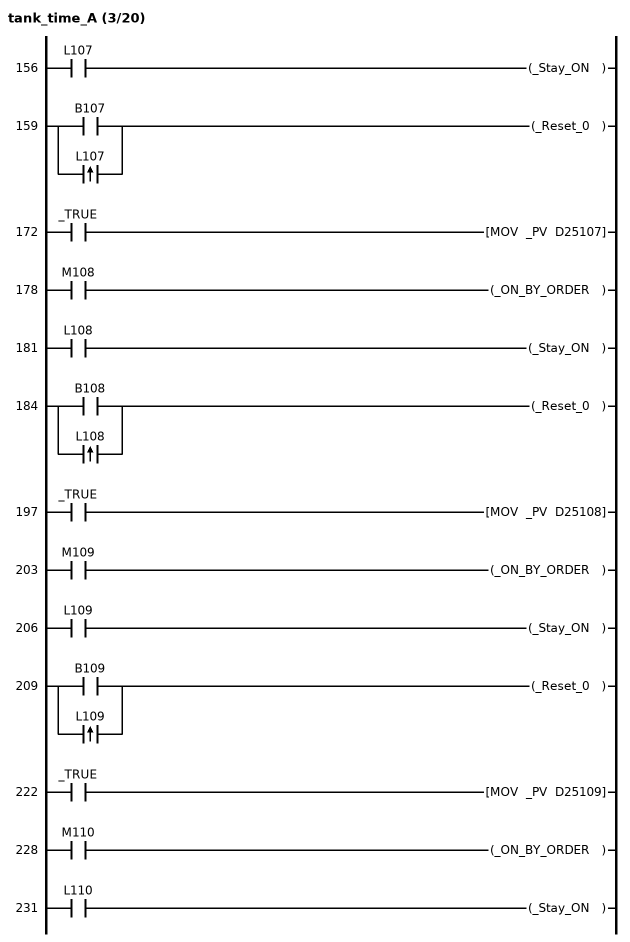
[picture p216: ladder of tank_time_A, rungs at steps 156 to 231]
156   LD      L107
      OUT     _Stay_ON
159   LD      B107
      ORP     L107
      OUT     _Reset_0
; FB START
; FB_NAME tank_PV
; INSTANCE_NAME tank_PV_7
; FB IN_B:ON_BY_ORDER
; FB OUT_PV:W
; FB IN_B:Stay_ON
; FB IN_B:Reset_0
; FB END
172   LD      _TRUE
      MOV     _PV D25107
; FB BLK END
; FB BLK START tank_PV(tank_PV_8)
178   LD      M108
      OUT     _ON_BY_ORDER
181   LD      L108
      OUT     _Stay_ON
184   LD      B108
      ORP     L108
      OUT     _Reset_0
; FB START
; FB_NAME tank_PV
; INSTANCE_NAME tank_PV_8
; FB IN_B:ON_BY_ORDER
; FB OUT_PV:W
; FB IN_B:Stay_ON
; FB IN_B:Reset_0
; FB END
197   LD      _TRUE
      MOV     _PV D25108
; FB BLK END
; FB BLK START tank_PV(tank_PV_9)
203   LD      M109
      OUT     _ON_BY_ORDER
206   LD      L109
      OUT     _Stay_ON
209   LD      B109
      ORP     L109
      OUT     _Reset_0
; FB START
; FB_NAME tank_PV
; INSTANCE_NAME tank_PV_9
; FB IN_B:ON_BY_ORDER
; FB OUT_PV:W
; FB IN_B:Stay_ON
; FB IN_B:Reset_0
; FB END
222   LD      _TRUE
      MOV     _PV D25109
; FB BLK END
; FB BLK START tank_PV(tank_PV_10)
228   LD      M110
      OUT     _ON_BY_ORDER
231   LD      L110
      OUT     _Stay_ON
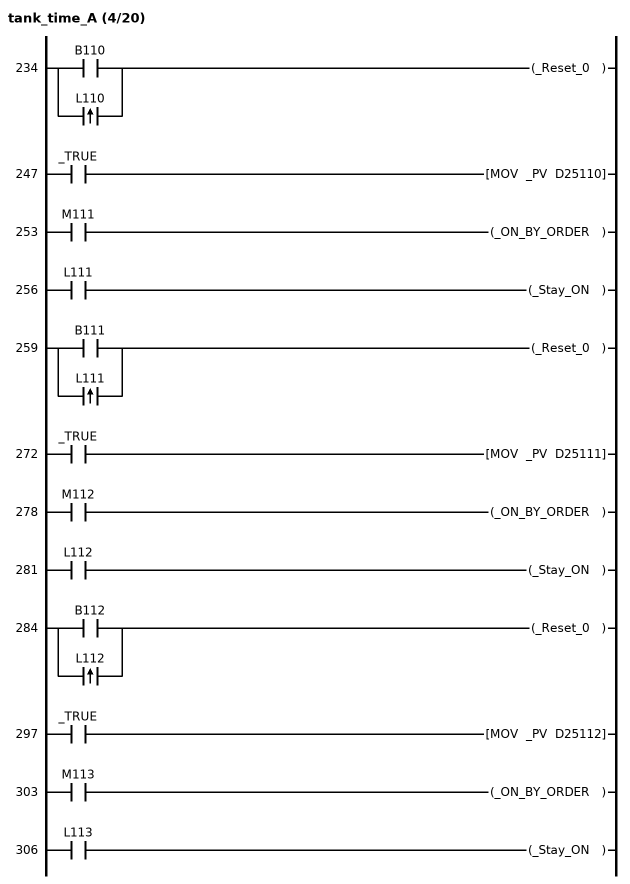
234   LD      B110
      ORP     L110
      OUT     _Reset_0
; FB START
; FB_NAME tank_PV
; INSTANCE_NAME tank_PV_10
; FB IN_B:ON_BY_ORDER
; FB OUT_PV:W
; FB IN_B:Stay_ON
; FB IN_B:Reset_0
; FB END
247   LD      _TRUE
      MOV     _PV D25110
; FB BLK END
; FB BLK START tank_PV(tank_PV_11)
253   LD      M111
      OUT     _ON_BY_ORDER
256   LD      L111
      OUT     _Stay_ON
259   LD      B111
      ORP     L111
      OUT     _Reset_0
; FB START
; FB_NAME tank_PV
; INSTANCE_NAME tank_PV_11
; FB IN_B:ON_BY_ORDER
; FB OUT_PV:W
; FB IN_B:Stay_ON
; FB IN_B:Reset_0
; FB END
272   LD      _TRUE
      MOV     _PV D25111
; FB BLK END
; FB BLK START tank_PV(tank_PV_12)
278   LD      M112
      OUT     _ON_BY_ORDER
281   LD      L112
      OUT     _Stay_ON
284   LD      B112
      ORP     L112
      OUT     _Reset_0
; FB START
; FB_NAME tank_PV
; INSTANCE_NAME tank_PV_12
; FB IN_B:ON_BY_ORDER
; FB OUT_PV:W
; FB IN_B:Stay_ON
; FB IN_B:Reset_0
; FB END
297   LD      _TRUE
      MOV     _PV D25112
; FB BLK END
; FB BLK START tank_PV(tank_PV_13)
303   LD      M113
      OUT     _ON_BY_ORDER
306   LD      L113
      OUT     _Stay_ON
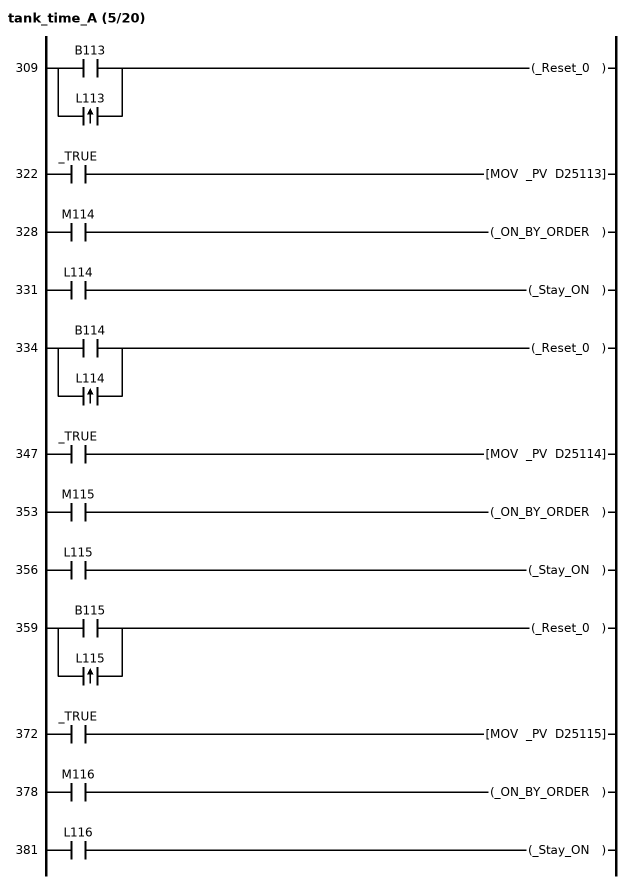
309   LD      B113
      ORP     L113
      OUT     _Reset_0
; FB START
; FB_NAME tank_PV
; INSTANCE_NAME tank_PV_13
; FB IN_B:ON_BY_ORDER
; FB OUT_PV:W
; FB IN_B:Stay_ON
; FB IN_B:Reset_0
; FB END
322   LD      _TRUE
      MOV     _PV D25113
; FB BLK END
; FB BLK START tank_PV(tank_PV_14)
328   LD      M114
      OUT     _ON_BY_ORDER
331   LD      L114
      OUT     _Stay_ON
334   LD      B114
      ORP     L114
      OUT     _Reset_0
; FB START
; FB_NAME tank_PV
; INSTANCE_NAME tank_PV_14
; FB IN_B:ON_BY_ORDER
; FB OUT_PV:W
; FB IN_B:Stay_ON
; FB IN_B:Reset_0
; FB END
347   LD      _TRUE
      MOV     _PV D25114
; FB BLK END
; FB BLK START tank_PV(tank_PV_15)
353   LD      M115
      OUT     _ON_BY_ORDER
356   LD      L115
      OUT     _Stay_ON
359   LD      B115
      ORP     L115
      OUT     _Reset_0
; FB START
; FB_NAME tank_PV
; INSTANCE_NAME tank_PV_15
; FB IN_B:ON_BY_ORDER
; FB OUT_PV:W
; FB IN_B:Stay_ON
; FB IN_B:Reset_0
; FB END
372   LD      _TRUE
      MOV     _PV D25115
; FB BLK END
; FB BLK START tank_PV(tank_PV_16)
378   LD      M116
      OUT     _ON_BY_ORDER
381   LD      L116
      OUT     _Stay_ON
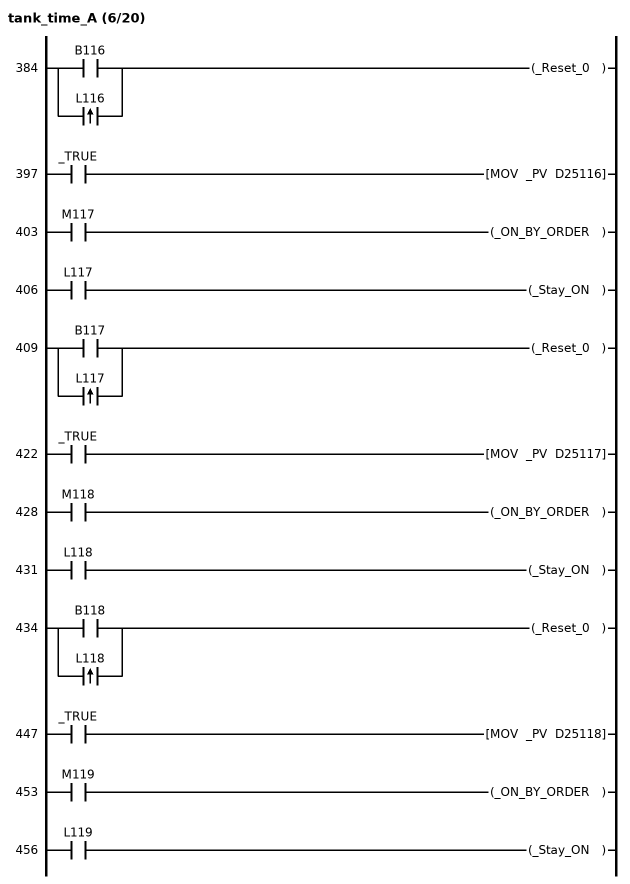
384   LD      B116
      ORP     L116
      OUT     _Reset_0
; FB START
; FB_NAME tank_PV
; INSTANCE_NAME tank_PV_16
; FB IN_B:ON_BY_ORDER
; FB OUT_PV:W
; FB IN_B:Stay_ON
; FB IN_B:Reset_0
; FB END
397   LD      _TRUE
      MOV     _PV D25116
; FB BLK END
; FB BLK START tank_PV(tank_PV_17)
403   LD      M117
      OUT     _ON_BY_ORDER
406   LD      L117
      OUT     _Stay_ON
409   LD      B117
      ORP     L117
      OUT     _Reset_0
; FB START
; FB_NAME tank_PV
; INSTANCE_NAME tank_PV_17
; FB IN_B:ON_BY_ORDER
; FB OUT_PV:W
; FB IN_B:Stay_ON
; FB IN_B:Reset_0
; FB END
422   LD      _TRUE
      MOV     _PV D25117
; FB BLK END
; FB BLK START tank_PV(tank_PV_18)
428   LD      M118
      OUT     _ON_BY_ORDER
431   LD      L118
      OUT     _Stay_ON
434   LD      B118
      ORP     L118
      OUT     _Reset_0
; FB START
; FB_NAME tank_PV
; INSTANCE_NAME tank_PV_18
; FB IN_B:ON_BY_ORDER
; FB OUT_PV:W
; FB IN_B:Stay_ON
; FB IN_B:Reset_0
; FB END
447   LD      _TRUE
      MOV     _PV D25118
; FB BLK END
; FB BLK START tank_PV(tank_PV_19)
453   LD      M119
      OUT     _ON_BY_ORDER
456   LD      L119
      OUT     _Stay_ON
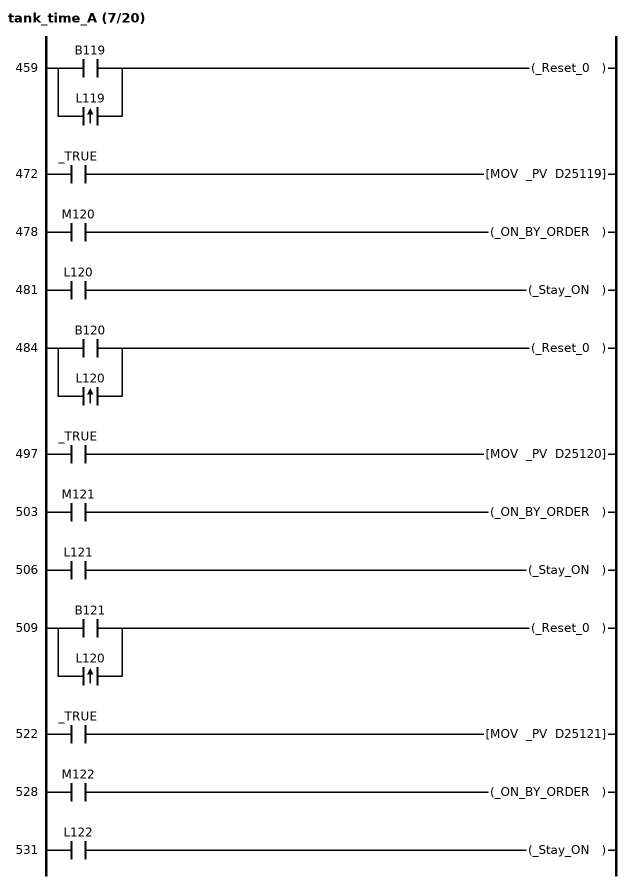
459   LD      B119
      ORP     L119
      OUT     _Reset_0
; FB START
; FB_NAME tank_PV
; INSTANCE_NAME tank_PV_19
; FB IN_B:ON_BY_ORDER
; FB OUT_PV:W
; FB IN_B:Stay_ON
; FB IN_B:Reset_0
; FB END
472   LD      _TRUE
      MOV     _PV D25119
; FB BLK END
; FB BLK START tank_PV(tank_PV_20)
478   LD      M120
      OUT     _ON_BY_ORDER
481   LD      L120
      OUT     _Stay_ON
484   LD      B120
      ORP     L120
      OUT     _Reset_0
; FB START
; FB_NAME tank_PV
; INSTANCE_NAME tank_PV_20
; FB IN_B:ON_BY_ORDER
; FB OUT_PV:W
; FB IN_B:Stay_ON
; FB IN_B:Reset_0
; FB END
497   LD      _TRUE
      MOV     _PV D25120
; FB BLK END
; FB BLK START tank_PV(tank_PV_21)
503   LD      M121
      OUT     _ON_BY_ORDER
506   LD      L121
      OUT     _Stay_ON
509   LD      B121
      ORP     L120
      OUT     _Reset_0
; FB START
; FB_NAME tank_PV
; INSTANCE_NAME tank_PV_21
; FB IN_B:ON_BY_ORDER
; FB OUT_PV:W
; FB IN_B:Stay_ON
; FB IN_B:Reset_0
; FB END
522   LD      _TRUE
      MOV     _PV D25121
; FB BLK END
; FB BLK START tank_PV(tank_PV_22)
528   LD      M122
      OUT     _ON_BY_ORDER
531   LD      L122
      OUT     _Stay_ON
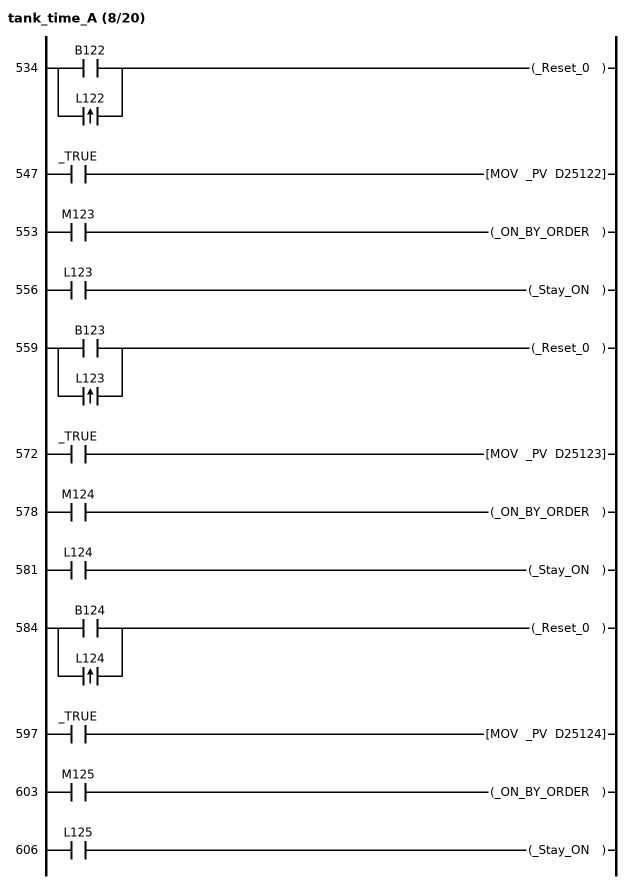
534   LD      B122
      ORP     L122
      OUT     _Reset_0
; FB START
; FB_NAME tank_PV
; INSTANCE_NAME tank_PV_22
; FB IN_B:ON_BY_ORDER
; FB OUT_PV:W
; FB IN_B:Stay_ON
; FB IN_B:Reset_0
; FB END
547   LD      _TRUE
      MOV     _PV D25122
; FB BLK END
; FB BLK START tank_PV(tank_PV_23)
553   LD      M123
      OUT     _ON_BY_ORDER
556   LD      L123
      OUT     _Stay_ON
559   LD      B123
      ORP     L123
      OUT     _Reset_0
; FB START
; FB_NAME tank_PV
; INSTANCE_NAME tank_PV_23
; FB IN_B:ON_BY_ORDER
; FB OUT_PV:W
; FB IN_B:Stay_ON
; FB IN_B:Reset_0
; FB END
572   LD      _TRUE
      MOV     _PV D25123
; FB BLK END
; FB BLK START tank_PV(tank_PV_24)
578   LD      M124
      OUT     _ON_BY_ORDER
581   LD      L124
      OUT     _Stay_ON
584   LD      B124
      ORP     L124
      OUT     _Reset_0
; FB START
; FB_NAME tank_PV
; INSTANCE_NAME tank_PV_24
; FB IN_B:ON_BY_ORDER
; FB OUT_PV:W
; FB IN_B:Stay_ON
; FB IN_B:Reset_0
; FB END
597   LD      _TRUE
      MOV     _PV D25124
; FB BLK END
; FB BLK START tank_PV(tank_PV_25)
603   LD      M125
      OUT     _ON_BY_ORDER
606   LD      L125
      OUT     _Stay_ON
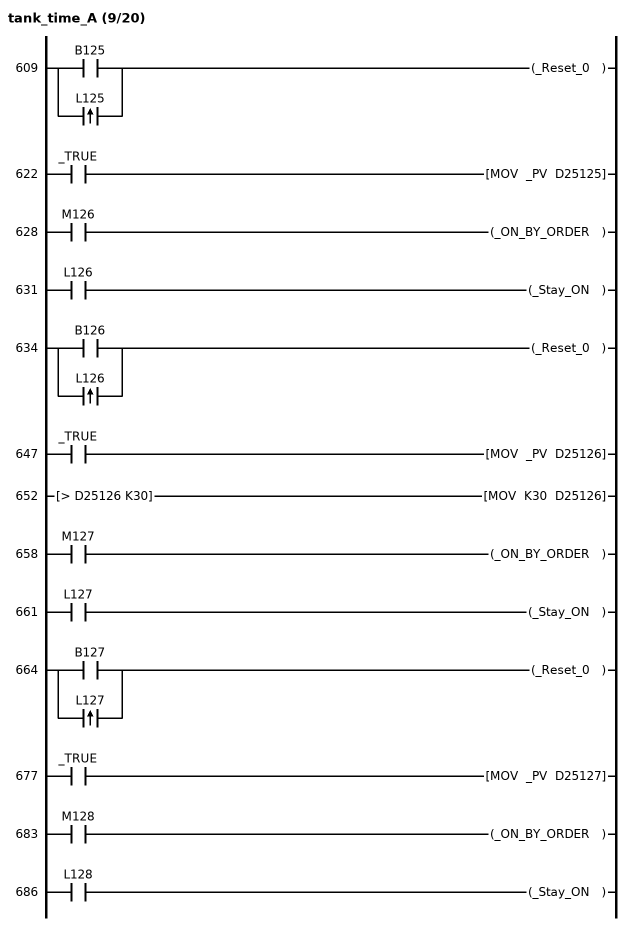
609   LD      B125
      ORP     L125
      OUT     _Reset_0
; FB START
; FB_NAME tank_PV
; INSTANCE_NAME tank_PV_25
; FB IN_B:ON_BY_ORDER
; FB OUT_PV:W
; FB IN_B:Stay_ON
; FB IN_B:Reset_0
; FB END
622   LD      _TRUE
      MOV     _PV D25125
; FB BLK END
; FB BLK START tank_PV(tank_PV_26)
628   LD      M126
      OUT     _ON_BY_ORDER
631   LD      L126
      OUT     _Stay_ON
634   LD      B126
      ORP     L126
      OUT     _Reset_0
; FB START
; FB_NAME tank_PV
; INSTANCE_NAME tank_PV_26
; FB IN_B:ON_BY_ORDER
; FB OUT_PV:W
; FB IN_B:Stay_ON
; FB IN_B:Reset_0
; FB END
647   LD      _TRUE
      MOV     _PV D25126
; FB BLK END
652   LD>     D25126 K30
      MOV     K30 D25126
; FB BLK START tank_PV(tank_PV_27)
658   LD      M127
      OUT     _ON_BY_ORDER
661   LD      L127
      OUT     _Stay_ON
664   LD      B127
      ORP     L127
      OUT     _Reset_0
; FB START
; FB_NAME tank_PV
; INSTANCE_NAME tank_PV_27
; FB IN_B:ON_BY_ORDER
; FB OUT_PV:W
; FB IN_B:Stay_ON
; FB IN_B:Reset_0
; FB END
677   LD      _TRUE
      MOV     _PV D25127
; FB BLK END
; FB BLK START tank_PV(tank_PV_28)
683   LD      M128
      OUT     _ON_BY_ORDER
686   LD      L128
      OUT     _Stay_ON
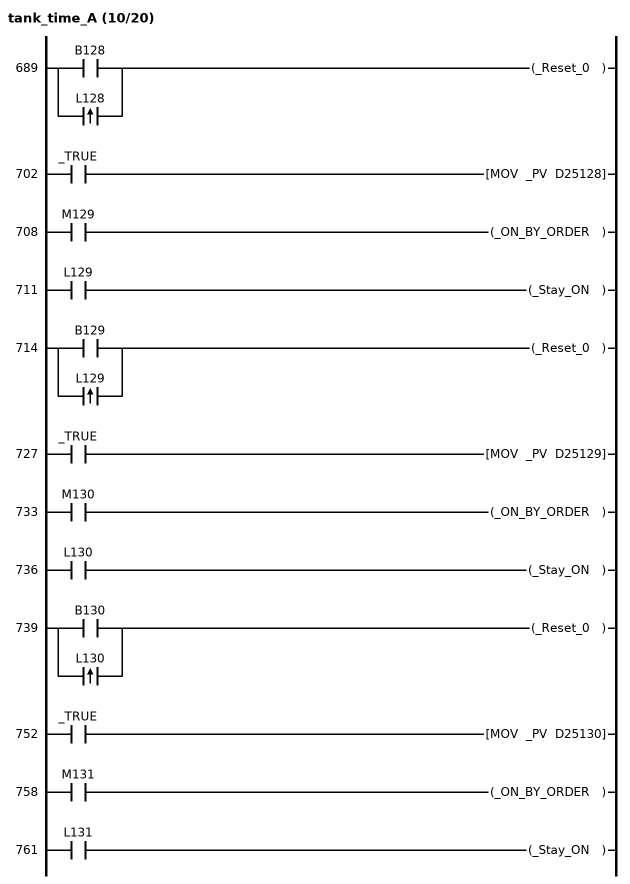
689   LD      B128
      ORP     L128
      OUT     _Reset_0
; FB START
; FB_NAME tank_PV
; INSTANCE_NAME tank_PV_28
; FB IN_B:ON_BY_ORDER
; FB OUT_PV:W
; FB IN_B:Stay_ON
; FB IN_B:Reset_0
; FB END
702   LD      _TRUE
      MOV     _PV D25128
; FB BLK END
; FB BLK START tank_PV(tank_PV_29)
708   LD      M129
      OUT     _ON_BY_ORDER
711   LD      L129
      OUT     _Stay_ON
714   LD      B129
      ORP     L129
      OUT     _Reset_0
; FB START
; FB_NAME tank_PV
; INSTANCE_NAME tank_PV_29
; FB IN_B:ON_BY_ORDER
; FB OUT_PV:W
; FB IN_B:Stay_ON
; FB IN_B:Reset_0
; FB END
727   LD      _TRUE
      MOV     _PV D25129
; FB BLK END
; FB BLK START tank_PV(tank_PV_30)
733   LD      M130
      OUT     _ON_BY_ORDER
736   LD      L130
      OUT     _Stay_ON
739   LD      B130
      ORP     L130
      OUT     _Reset_0
; FB START
; FB_NAME tank_PV
; INSTANCE_NAME tank_PV_30
; FB IN_B:ON_BY_ORDER
; FB OUT_PV:W
; FB IN_B:Stay_ON
; FB IN_B:Reset_0
; FB END
752   LD      _TRUE
      MOV     _PV D25130
; FB BLK END
; FB BLK START tank_PV(tank_PV_31)
758   LD      M131
      OUT     _ON_BY_ORDER
761   LD      L131
      OUT     _Stay_ON
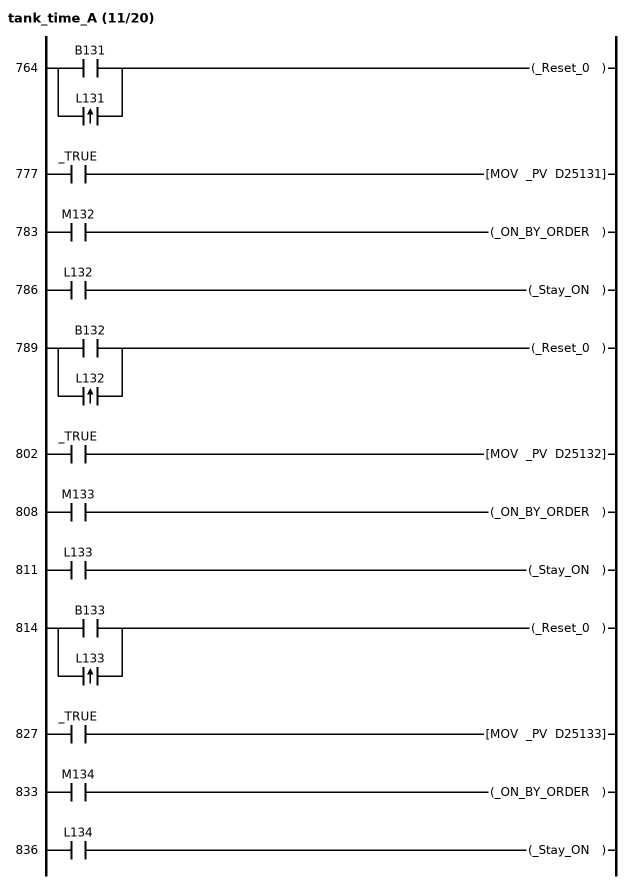
764   LD      B131
      ORP     L131
      OUT     _Reset_0
; FB START
; FB_NAME tank_PV
; INSTANCE_NAME tank_PV_31
; FB IN_B:ON_BY_ORDER
; FB OUT_PV:W
; FB IN_B:Stay_ON
; FB IN_B:Reset_0
; FB END
777   LD      _TRUE
      MOV     _PV D25131
; FB BLK END
; FB BLK START tank_PV(tank_PV_32)
783   LD      M132
      OUT     _ON_BY_ORDER
786   LD      L132
      OUT     _Stay_ON
789   LD      B132
      ORP     L132
      OUT     _Reset_0
; FB START
; FB_NAME tank_PV
; INSTANCE_NAME tank_PV_32
; FB IN_B:ON_BY_ORDER
; FB OUT_PV:W
; FB IN_B:Stay_ON
; FB IN_B:Reset_0
; FB END
802   LD      _TRUE
      MOV     _PV D25132
; FB BLK END
; FB BLK START tank_PV(tank_PV_33)
808   LD      M133
      OUT     _ON_BY_ORDER
811   LD      L133
      OUT     _Stay_ON
814   LD      B133
      ORP     L133
      OUT     _Reset_0
; FB START
; FB_NAME tank_PV
; INSTANCE_NAME tank_PV_33
; FB IN_B:ON_BY_ORDER
; FB OUT_PV:W
; FB IN_B:Stay_ON
; FB IN_B:Reset_0
; FB END
827   LD      _TRUE
      MOV     _PV D25133
; FB BLK END
; FB BLK START tank_PV(tank_PV_34)
833   LD      M134
      OUT     _ON_BY_ORDER
836   LD      L134
      OUT     _Stay_ON
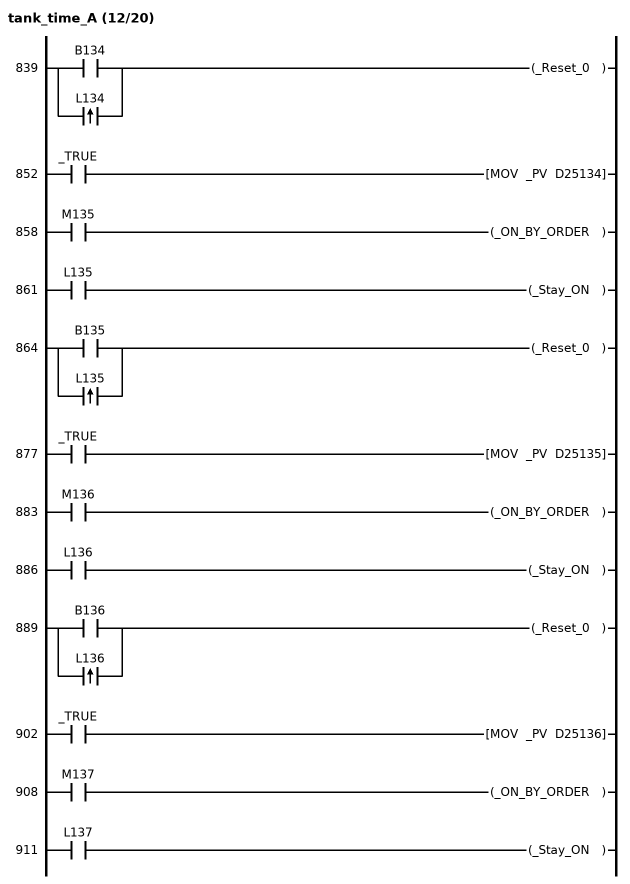
839   LD      B134
      ORP     L134
      OUT     _Reset_0
; FB START
; FB_NAME tank_PV
; INSTANCE_NAME tank_PV_34
; FB IN_B:ON_BY_ORDER
; FB OUT_PV:W
; FB IN_B:Stay_ON
; FB IN_B:Reset_0
; FB END
852   LD      _TRUE
      MOV     _PV D25134
; FB BLK END
; FB BLK START tank_PV(tank_PV_35)
858   LD      M135
      OUT     _ON_BY_ORDER
861   LD      L135
      OUT     _Stay_ON
864   LD      B135
      ORP     L135
      OUT     _Reset_0
; FB START
; FB_NAME tank_PV
; INSTANCE_NAME tank_PV_35
; FB IN_B:ON_BY_ORDER
; FB OUT_PV:W
; FB IN_B:Stay_ON
; FB IN_B:Reset_0
; FB END
877   LD      _TRUE
      MOV     _PV D25135
; FB BLK END
; FB BLK START tank_PV(tank_PV_36)
883   LD      M136
      OUT     _ON_BY_ORDER
886   LD      L136
      OUT     _Stay_ON
889   LD      B136
      ORP     L136
      OUT     _Reset_0
; FB START
; FB_NAME tank_PV
; INSTANCE_NAME tank_PV_36
; FB IN_B:ON_BY_ORDER
; FB OUT_PV:W
; FB IN_B:Stay_ON
; FB IN_B:Reset_0
; FB END
902   LD      _TRUE
      MOV     _PV D25136
; FB BLK END
; FB BLK START tank_PV(tank_PV_37)
908   LD      M137
      OUT     _ON_BY_ORDER
911   LD      L137
      OUT     _Stay_ON
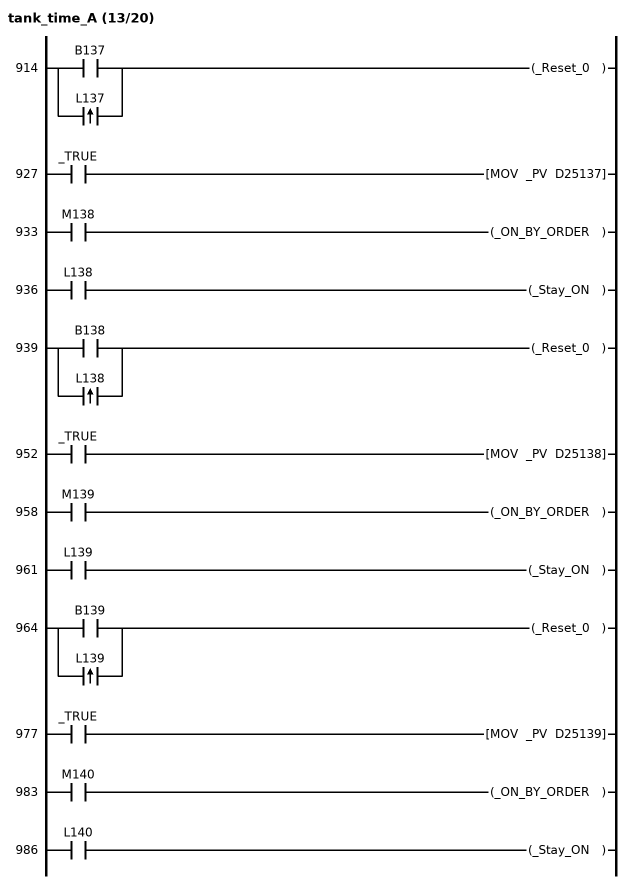
914   LD      B137
      ORP     L137
      OUT     _Reset_0
; FB START
; FB_NAME tank_PV
; INSTANCE_NAME tank_PV_37
; FB IN_B:ON_BY_ORDER
; FB OUT_PV:W
; FB IN_B:Stay_ON
; FB IN_B:Reset_0
; FB END
927   LD      _TRUE
      MOV     _PV D25137
; FB BLK END
; FB BLK START tank_PV(tank_PV_38)
933   LD      M138
      OUT     _ON_BY_ORDER
936   LD      L138
      OUT     _Stay_ON
939   LD      B138
      ORP     L138
      OUT     _Reset_0
; FB START
; FB_NAME tank_PV
; INSTANCE_NAME tank_PV_38
; FB IN_B:ON_BY_ORDER
; FB OUT_PV:W
; FB IN_B:Stay_ON
; FB IN_B:Reset_0
; FB END
952   LD      _TRUE
      MOV     _PV D25138
; FB BLK END
; FB BLK START tank_PV(tank_PV_39)
958   LD      M139
      OUT     _ON_BY_ORDER
961   LD      L139
      OUT     _Stay_ON
964   LD      B139
      ORP     L139
      OUT     _Reset_0
; FB START
; FB_NAME tank_PV
; INSTANCE_NAME tank_PV_39
; FB IN_B:ON_BY_ORDER
; FB OUT_PV:W
; FB IN_B:Stay_ON
; FB IN_B:Reset_0
; FB END
977   LD      _TRUE
      MOV     _PV D25139
; FB BLK END
; FB BLK START tank_PV(tank_PV_40)
983   LD      M140
      OUT     _ON_BY_ORDER
986   LD      L140
      OUT     _Stay_ON
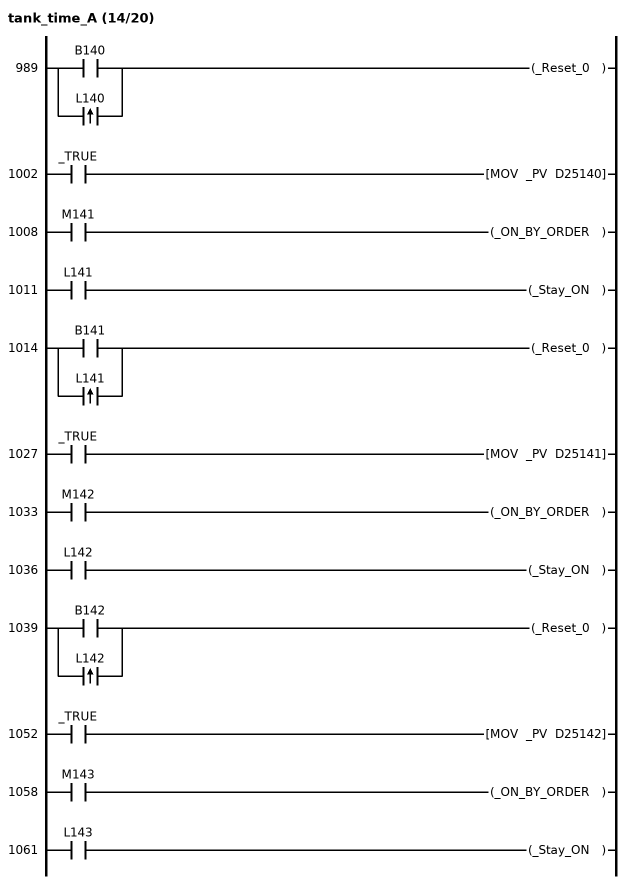
989   LD      B140
      ORP     L140
      OUT     _Reset_0
; FB START
; FB_NAME tank_PV
; INSTANCE_NAME tank_PV_40
; FB IN_B:ON_BY_ORDER
; FB OUT_PV:W
; FB IN_B:Stay_ON
; FB IN_B:Reset_0
; FB END
1002  LD      _TRUE
      MOV     _PV D25140
; FB BLK END
; FB BLK START tank_PV(tank_PV_41)
1008  LD      M141
      OUT     _ON_BY_ORDER
1011  LD      L141
      OUT     _Stay_ON
1014  LD      B141
      ORP     L141
      OUT     _Reset_0
; FB START
; FB_NAME tank_PV
; INSTANCE_NAME tank_PV_41
; FB IN_B:ON_BY_ORDER
; FB OUT_PV:W
; FB IN_B:Stay_ON
; FB IN_B:Reset_0
; FB END
1027  LD      _TRUE
      MOV     _PV D25141
; FB BLK END
; FB BLK START tank_PV(tank_PV_42)
1033  LD      M142
      OUT     _ON_BY_ORDER
1036  LD      L142
      OUT     _Stay_ON
1039  LD      B142
      ORP     L142
      OUT     _Reset_0
; FB START
; FB_NAME tank_PV
; INSTANCE_NAME tank_PV_42
; FB IN_B:ON_BY_ORDER
; FB OUT_PV:W
; FB IN_B:Stay_ON
; FB IN_B:Reset_0
; FB END
1052  LD      _TRUE
      MOV     _PV D25142
; FB BLK END
; FB BLK START tank_PV(tank_PV_43)
1058  LD      M143
      OUT     _ON_BY_ORDER
1061  LD      L143
      OUT     _Stay_ON
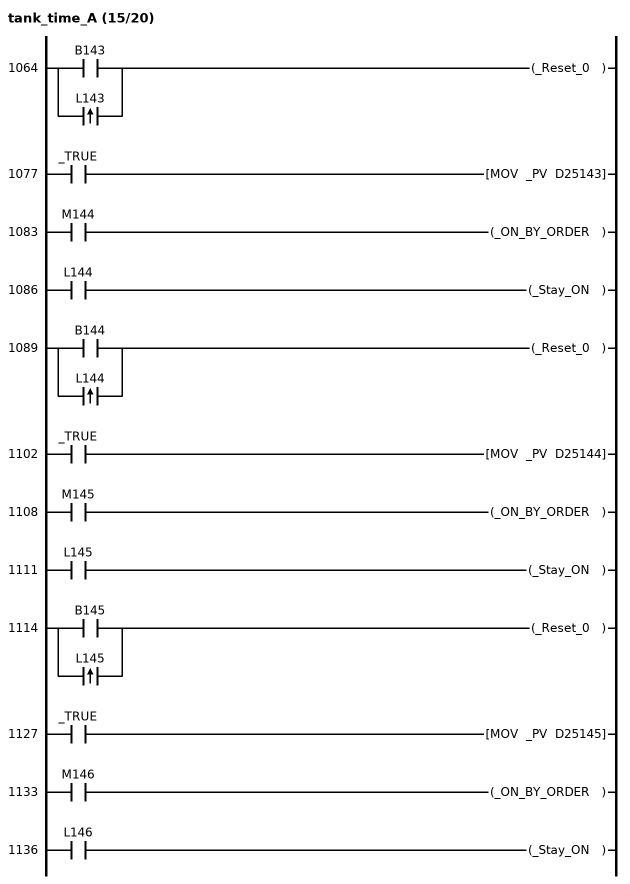
1064  LD      B143
      ORP     L143
      OUT     _Reset_0
; FB START
; FB_NAME tank_PV
; INSTANCE_NAME tank_PV_43
; FB IN_B:ON_BY_ORDER
; FB OUT_PV:W
; FB IN_B:Stay_ON
; FB IN_B:Reset_0
; FB END
1077  LD      _TRUE
      MOV     _PV D25143
; FB BLK END
; FB BLK START tank_PV(tank_PV_44)
1083  LD      M144
      OUT     _ON_BY_ORDER
1086  LD      L144
      OUT     _Stay_ON
1089  LD      B144
      ORP     L144
      OUT     _Reset_0
; FB START
; FB_NAME tank_PV
; INSTANCE_NAME tank_PV_44
; FB IN_B:ON_BY_ORDER
; FB OUT_PV:W
; FB IN_B:Stay_ON
; FB IN_B:Reset_0
; FB END
1102  LD      _TRUE
      MOV     _PV D25144
; FB BLK END
; FB BLK START tank_PV(tank_PV_45)
1108  LD      M145
      OUT     _ON_BY_ORDER
1111  LD      L145
      OUT     _Stay_ON
1114  LD      B145
      ORP     L145
      OUT     _Reset_0
; FB START
; FB_NAME tank_PV
; INSTANCE_NAME tank_PV_45
; FB IN_B:ON_BY_ORDER
; FB OUT_PV:W
; FB IN_B:Stay_ON
; FB IN_B:Reset_0
; FB END
1127  LD      _TRUE
      MOV     _PV D25145
; FB BLK END
; FB BLK START tank_PV(tank_PV_46)
1133  LD      M146
      OUT     _ON_BY_ORDER
1136  LD      L146
      OUT     _Stay_ON
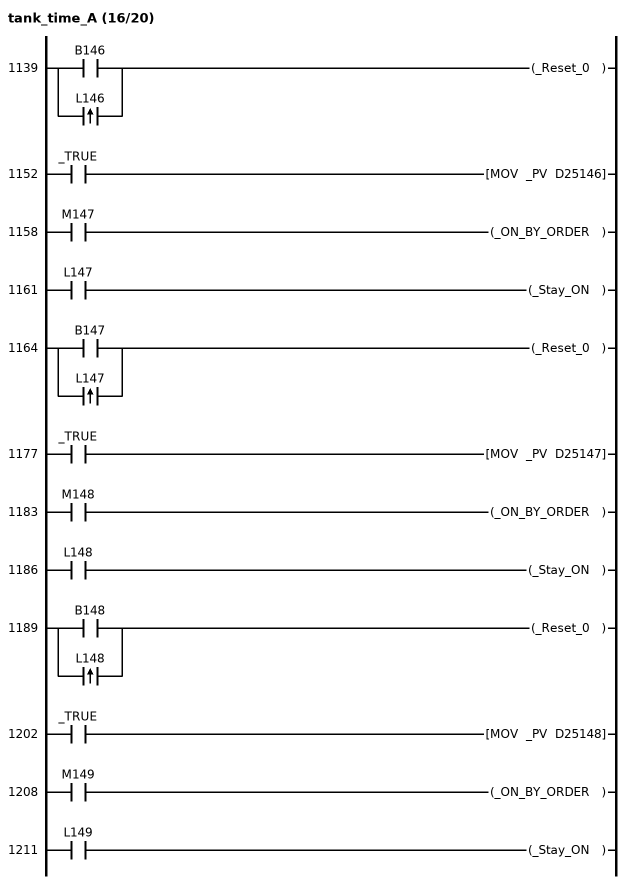
1139  LD      B146
      ORP     L146
      OUT     _Reset_0
; FB START
; FB_NAME tank_PV
; INSTANCE_NAME tank_PV_46
; FB IN_B:ON_BY_ORDER
; FB OUT_PV:W
; FB IN_B:Stay_ON
; FB IN_B:Reset_0
; FB END
1152  LD      _TRUE
      MOV     _PV D25146
; FB BLK END
; FB BLK START tank_PV(tank_PV_47)
1158  LD      M147
      OUT     _ON_BY_ORDER
1161  LD      L147
      OUT     _Stay_ON
1164  LD      B147
      ORP     L147
      OUT     _Reset_0
; FB START
; FB_NAME tank_PV
; INSTANCE_NAME tank_PV_47
; FB IN_B:ON_BY_ORDER
; FB OUT_PV:W
; FB IN_B:Stay_ON
; FB IN_B:Reset_0
; FB END
1177  LD      _TRUE
      MOV     _PV D25147
; FB BLK END
; FB BLK START tank_PV(tank_PV_48)
1183  LD      M148
      OUT     _ON_BY_ORDER
1186  LD      L148
      OUT     _Stay_ON
1189  LD      B148
      ORP     L148
      OUT     _Reset_0
; FB START
; FB_NAME tank_PV
; INSTANCE_NAME tank_PV_48
; FB IN_B:ON_BY_ORDER
; FB OUT_PV:W
; FB IN_B:Stay_ON
; FB IN_B:Reset_0
; FB END
1202  LD      _TRUE
      MOV     _PV D25148
; FB BLK END
; FB BLK START tank_PV(tank_PV_49)
1208  LD      M149
      OUT     _ON_BY_ORDER
1211  LD      L149
      OUT     _Stay_ON
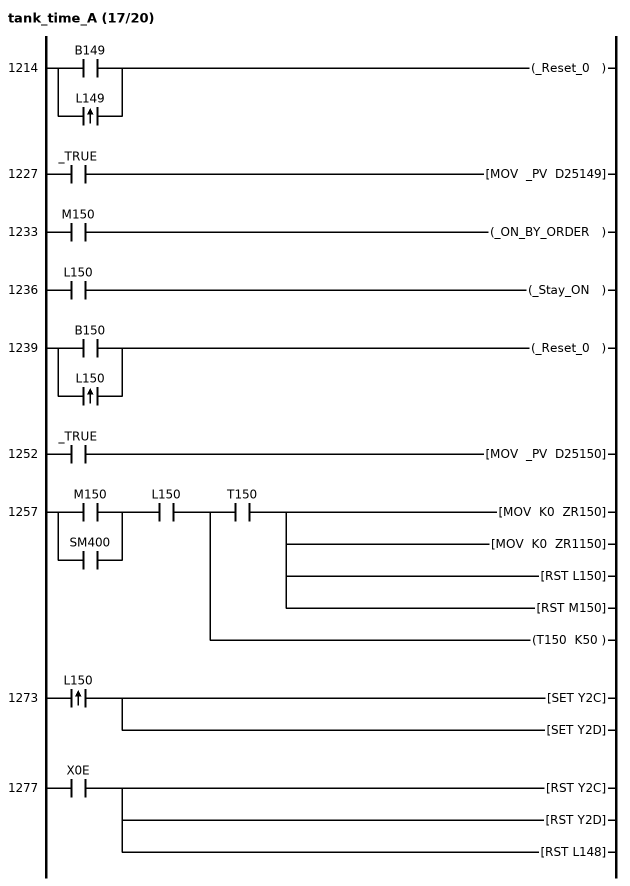
1214  LD      B149
      ORP     L149
      OUT     _Reset_0
; FB START
; FB_NAME tank_PV
; INSTANCE_NAME tank_PV_49
; FB IN_B:ON_BY_ORDER
; FB OUT_PV:W
; FB IN_B:Stay_ON
; FB IN_B:Reset_0
; FB END
1227  LD      _TRUE
      MOV     _PV D25149
; FB BLK END
; FB BLK START tank_PV(tank_PV_50)
1233  LD      M150
      OUT     _ON_BY_ORDER
1236  LD      L150
      OUT     _Stay_ON
1239  LD      B150
      ORP     L150
      OUT     _Reset_0
; FB START
; FB_NAME tank_PV
; INSTANCE_NAME tank_PV_50
; FB IN_B:ON_BY_ORDER
; FB OUT_PV:W
; FB IN_B:Stay_ON
; FB IN_B:Reset_0
; FB END
1252  LD      _TRUE
      MOV     _PV D25150
; FB BLK END
1257  LD      M150
      OR      SM400
      AND     L150
      MPS
      AND     T150
      MOV     K0 ZR150
      MOV     K0 ZR1150
      RST     L150
      RST     M150
      MPP
      OUT     T150 K50
1273  LDP     L150
      SET     Y2C
      SET     Y2D
1277  LD      X0E
      RST     Y2C
      RST     Y2D
      RST     L148
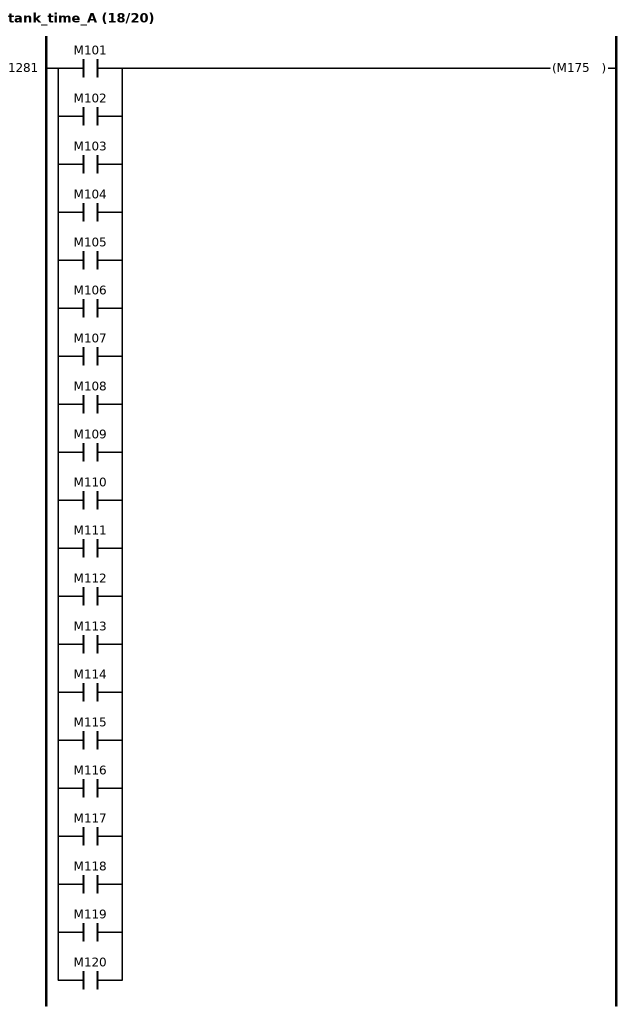
1281  LD      M101
      OR      M102
      OR      M103
      OR      M104
      OR      M105
      OR      M106
      OR      M107
      OR      M108
      OR      M109
      OR      M110
      OR      M111
      OR      M112
      OR      M113
      OR      M114
      OR      M115
      OR      M116
      OR      M117
      OR      M118
      OR      M119
      OR      M120
      OUT     M175
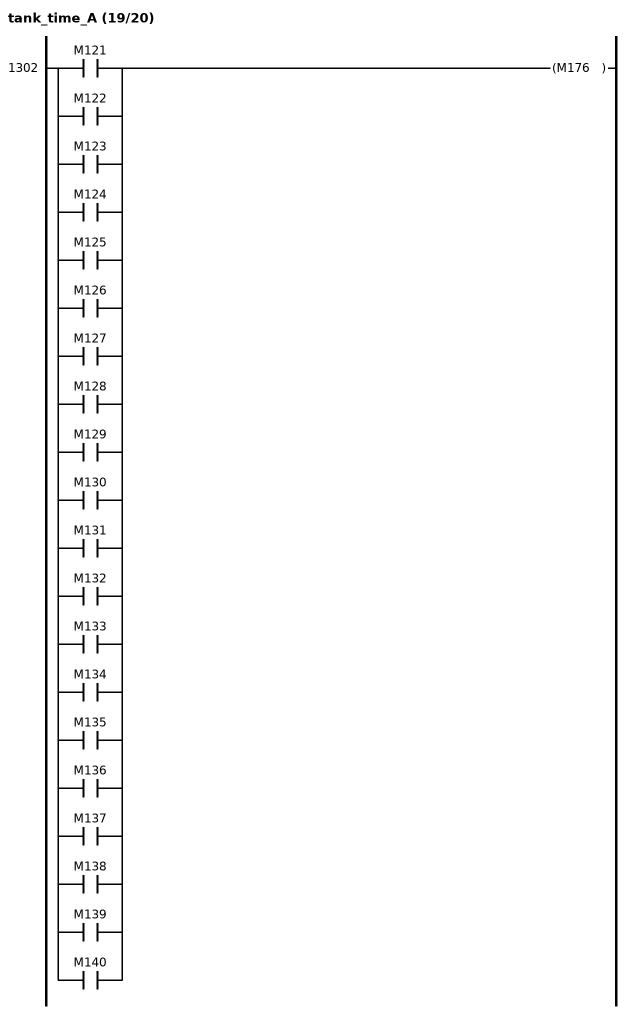
1302  LD      M121
      OR      M122
      OR      M123
      OR      M124
      OR      M125
      OR      M126
      OR      M127
      OR      M128
      OR      M129
      OR      M130
      OR      M131
      OR      M132
      OR      M133
      OR      M134
      OR      M135
      OR      M136
      OR      M137
      OR      M138
      OR      M139
      OR      M140
      OUT     M176
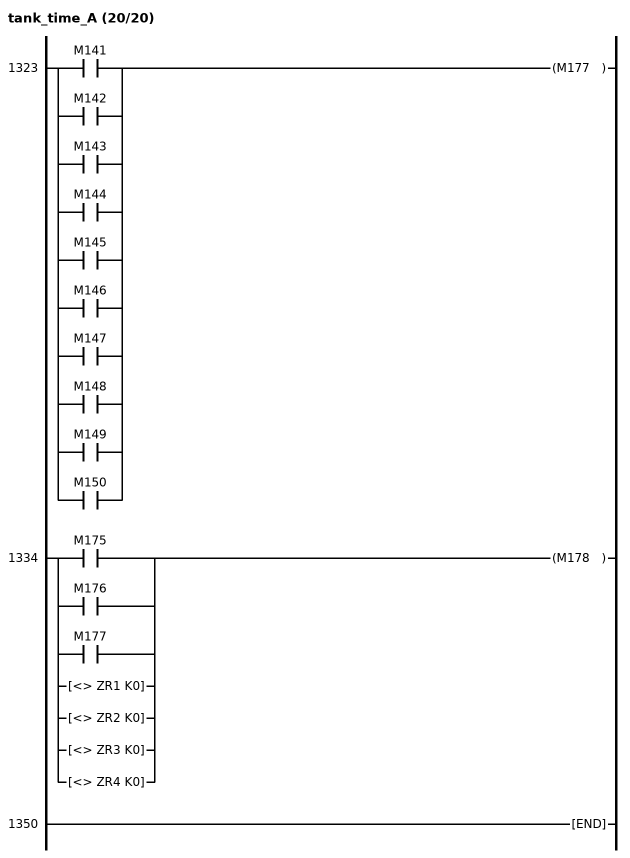
1323  LD      M141
      OR      M142
      OR      M143
      OR      M144
      OR      M145
      OR      M146
      OR      M147
      OR      M148
      OR      M149
      OR      M150
      OUT     M177
1334  LD      M175
      OR      M176
      OR      M177
      OR<>    ZR1 K0
      OR<>    ZR2 K0
      OR<>    ZR3 K0
      OR<>    ZR4 K0
      OUT     M178
1350  END
END_PROGRAM

PROGRAM temp_system
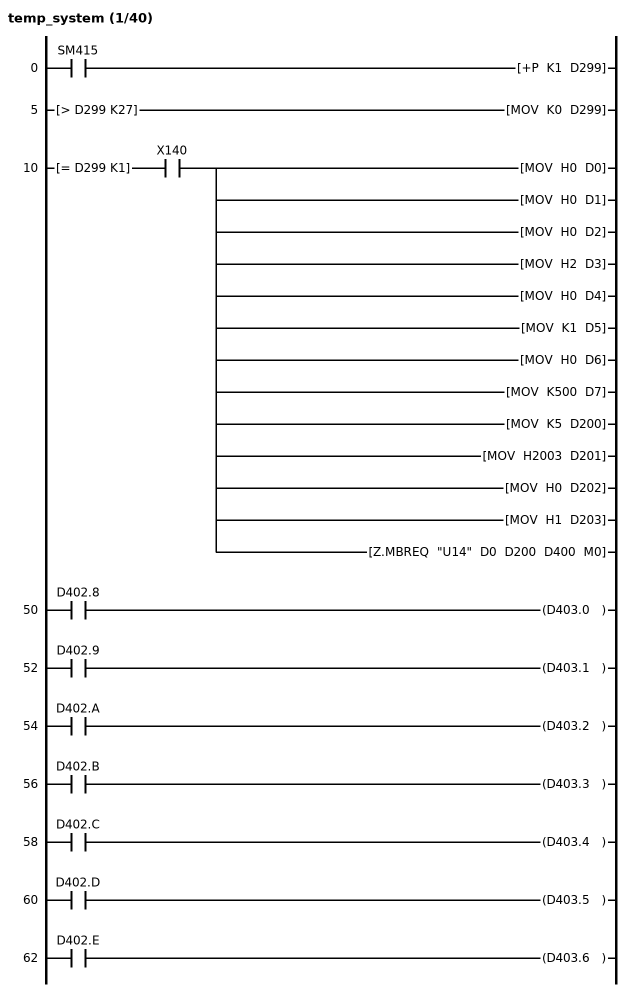
0     LD      SM415
      +P      K1 D299
5     LD>     D299 K27
      MOV     K0 D299
10    LD=     D299 K1
      AND     X140
      MOV     H0 D0
      MOV     H0 D1
      MOV     H0 D2
      MOV     H2 D3
      MOV     H0 D4
      MOV     K1 D5
      MOV     H0 D6
      MOV     K500 D7
      MOV     K5 D200
      MOV     H2003 D201
      MOV     H0 D202
      MOV     H1 D203
      Z.MBREQ "U14" D0 D200 D400 M0
50    LD      D402.8
      OUT     D403.0
52    LD      D402.9
      OUT     D403.1
54    LD      D402.A
      OUT     D403.2
56    LD      D402.B
      OUT     D403.3
58    LD      D402.C
      OUT     D403.4
60    LD      D402.D
      OUT     D403.5
62    LD      D402.E
      OUT     D403.6
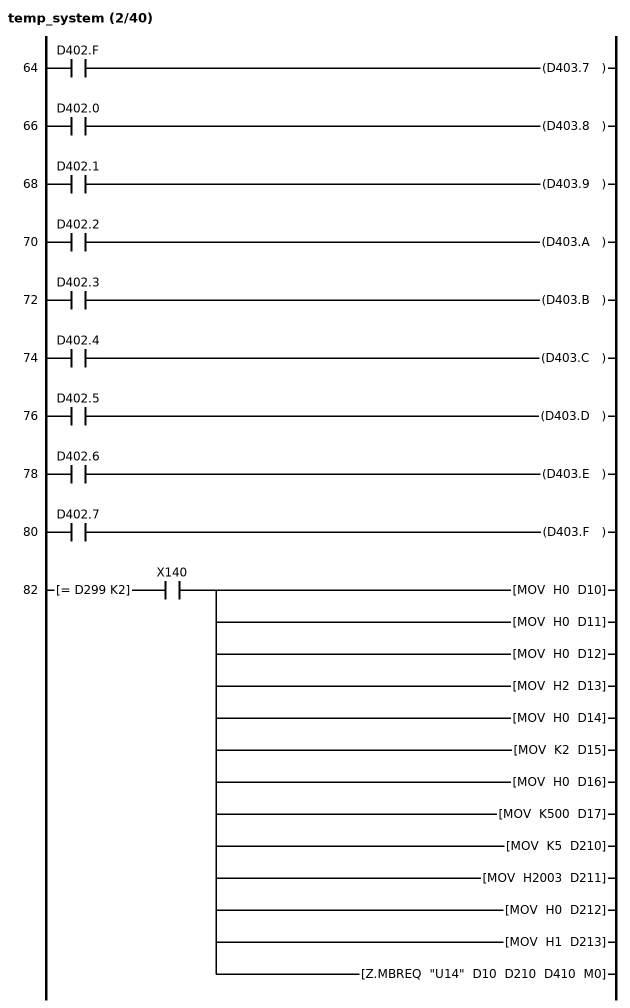
64    LD      D402.F
      OUT     D403.7
66    LD      D402.0
      OUT     D403.8
68    LD      D402.1
      OUT     D403.9
70    LD      D402.2
      OUT     D403.A
72    LD      D402.3
      OUT     D403.B
74    LD      D402.4
      OUT     D403.C
76    LD      D402.5
      OUT     D403.D
78    LD      D402.6
      OUT     D403.E
80    LD      D402.7
      OUT     D403.F
82    LD=     D299 K2
      AND     X140
      MOV     H0 D10
      MOV     H0 D11
      MOV     H0 D12
      MOV     H2 D13
      MOV     H0 D14
      MOV     K2 D15
      MOV     H0 D16
      MOV     K500 D17
      MOV     K5 D210
      MOV     H2003 D211
      MOV     H0 D212
      MOV     H1 D213
      Z.MBREQ "U14" D10 D210 D410 M0
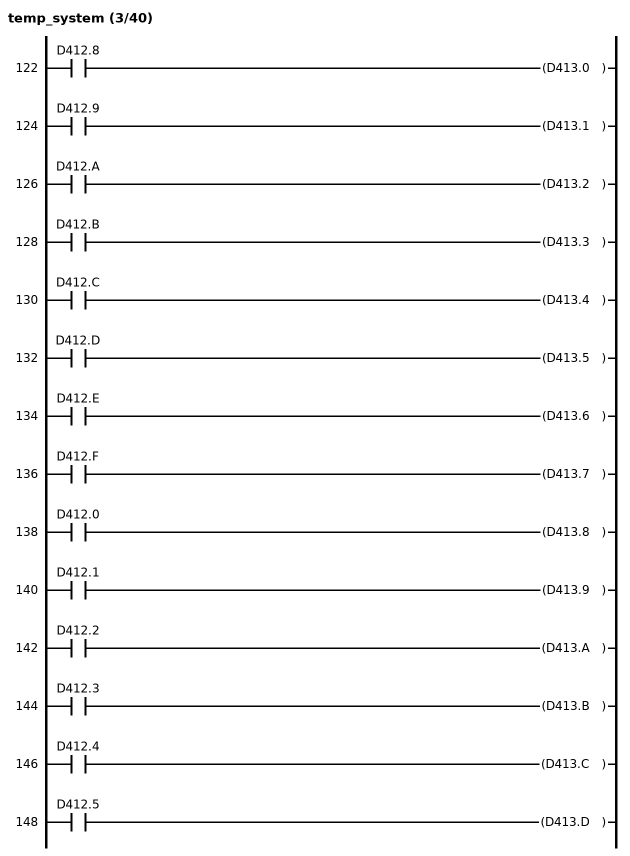
122   LD      D412.8
      OUT     D413.0
124   LD      D412.9
      OUT     D413.1
126   LD      D412.A
      OUT     D413.2
128   LD      D412.B
      OUT     D413.3
130   LD      D412.C
      OUT     D413.4
132   LD      D412.D
      OUT     D413.5
134   LD      D412.E
      OUT     D413.6
136   LD      D412.F
      OUT     D413.7
138   LD      D412.0
      OUT     D413.8
140   LD      D412.1
      OUT     D413.9
142   LD      D412.2
      OUT     D413.A
144   LD      D412.3
      OUT     D413.B
146   LD      D412.4
      OUT     D413.C
148   LD      D412.5
      OUT     D413.D
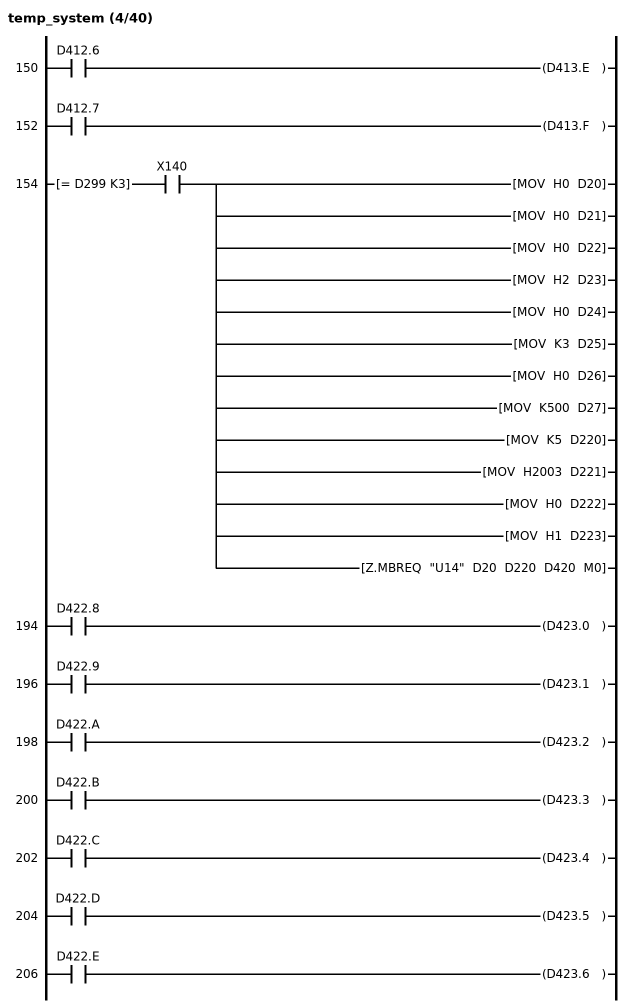
150   LD      D412.6
      OUT     D413.E
152   LD      D412.7
      OUT     D413.F
154   LD=     D299 K3
      AND     X140
      MOV     H0 D20
      MOV     H0 D21
      MOV     H0 D22
      MOV     H2 D23
      MOV     H0 D24
      MOV     K3 D25
      MOV     H0 D26
      MOV     K500 D27
      MOV     K5 D220
      MOV     H2003 D221
      MOV     H0 D222
      MOV     H1 D223
      Z.MBREQ "U14" D20 D220 D420 M0
194   LD      D422.8
      OUT     D423.0
196   LD      D422.9
      OUT     D423.1
198   LD      D422.A
      OUT     D423.2
200   LD      D422.B
      OUT     D423.3
202   LD      D422.C
      OUT     D423.4
204   LD      D422.D
      OUT     D423.5
206   LD      D422.E
      OUT     D423.6
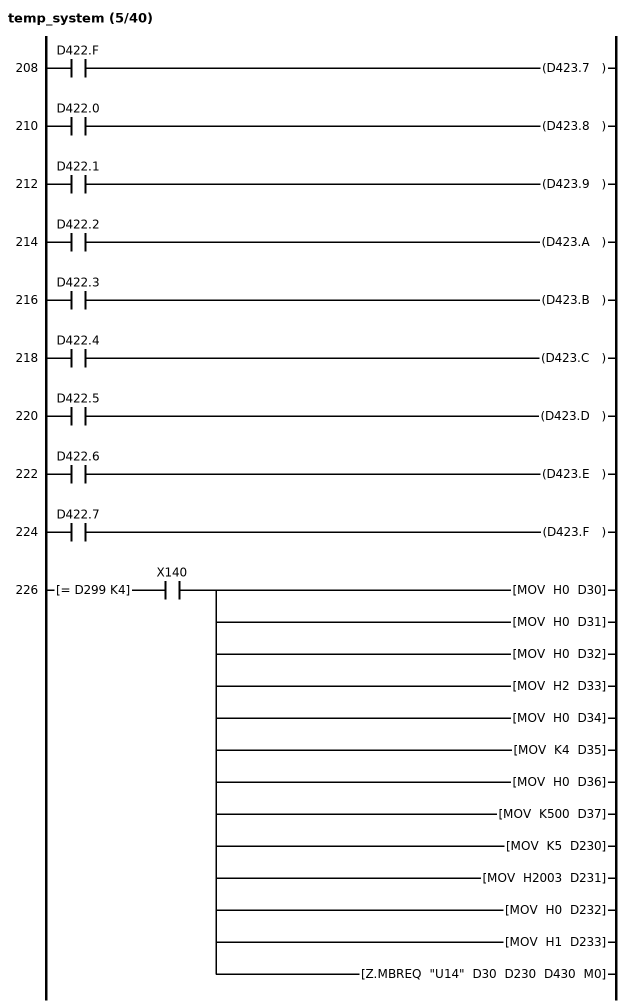
208   LD      D422.F
      OUT     D423.7
210   LD      D422.0
      OUT     D423.8
212   LD      D422.1
      OUT     D423.9
214   LD      D422.2
      OUT     D423.A
216   LD      D422.3
      OUT     D423.B
218   LD      D422.4
      OUT     D423.C
220   LD      D422.5
      OUT     D423.D
222   LD      D422.6
      OUT     D423.E
224   LD      D422.7
      OUT     D423.F
226   LD=     D299 K4
      AND     X140
      MOV     H0 D30
      MOV     H0 D31
      MOV     H0 D32
      MOV     H2 D33
      MOV     H0 D34
      MOV     K4 D35
      MOV     H0 D36
      MOV     K500 D37
      MOV     K5 D230
      MOV     H2003 D231
      MOV     H0 D232
      MOV     H1 D233
      Z.MBREQ "U14" D30 D230 D430 M0
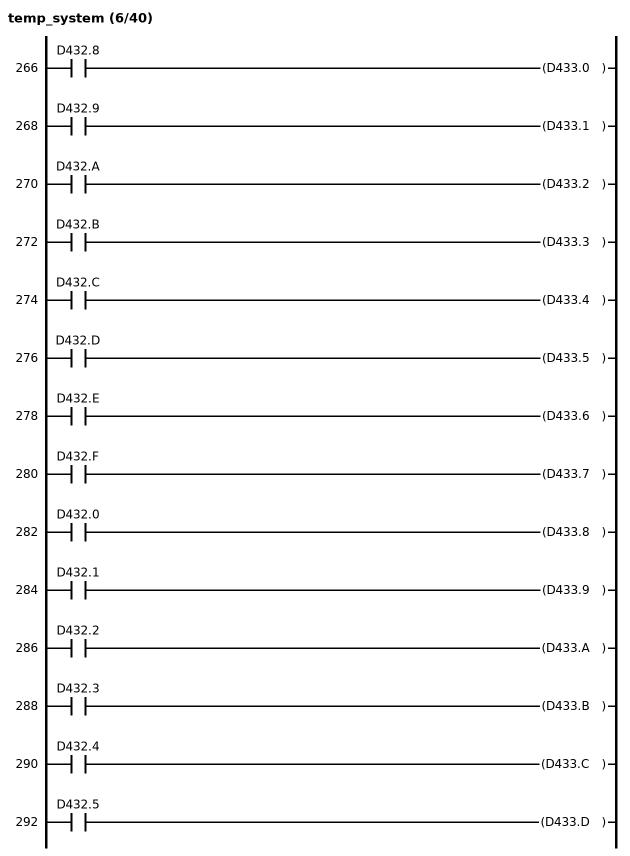
266   LD      D432.8
      OUT     D433.0
268   LD      D432.9
      OUT     D433.1
270   LD      D432.A
      OUT     D433.2
272   LD      D432.B
      OUT     D433.3
274   LD      D432.C
      OUT     D433.4
276   LD      D432.D
      OUT     D433.5
278   LD      D432.E
      OUT     D433.6
280   LD      D432.F
      OUT     D433.7
282   LD      D432.0
      OUT     D433.8
284   LD      D432.1
      OUT     D433.9
286   LD      D432.2
      OUT     D433.A
288   LD      D432.3
      OUT     D433.B
290   LD      D432.4
      OUT     D433.C
292   LD      D432.5
      OUT     D433.D
